INTERFACE I_AlarmControler

PROPERTY Active : REFERENCE TO BOOL
GET
END_GET
END_PROPERTY

PROPERTY ActiveCritical : REFERENCE TO UDINT
GET
END_GET
END_PROPERTY

PROPERTY ActiveError : REFERENCE TO UDINT
GET
END_GET
END_PROPERTY

PROPERTY ActiveInfo : REFERENCE TO UDINT
GET
END_GET
END_PROPERTY

PROPERTY ActiveVerbose : REFERENCE TO UDINT
GET
END_GET
END_PROPERTY

PROPERTY ActiveWarrning : REFERENCE TO UDINT
GET
END_GET
END_PROPERTY

PROPERTY Busy : REFERENCE TO BOOL
GET
END_GET
END_PROPERTY

PROPERTY Error : REFERENCE TO BOOL
GET
END_GET
END_PROPERTY

PROPERTY FileName : STRING
GET
END_GET
SET
END_SET
END_PROPERTY

PROPERTY MaxEvents : UDINT
GET
END_GET
END_PROPERTY

METHOD MR_Abort : BOOL
VAR_INPUT
END_VAR
END_METHOD

METHOD MR_Clear : BOOL
VAR_INPUT
	ipFilter : I_TcEventFilter;
	bResetConfirmation : BOOL;
END_VAR
END_METHOD

METHOD MR_ClearAll : BOOL
VAR_INPUT
	bResetConfirmation : BOOL;
END_VAR
END_METHOD

METHOD MR_Confirm : BOOL
VAR_INPUT
	ipFilter : I_TcEventFilter;
END_VAR
END_METHOD

METHOD MR_ConfirmAll : BOOL
VAR_INPUT
	bResetConfirmation : BOOL;
END_VAR
END_METHOD

METHOD MR_Export : BOOL
VAR_INPUT
END_VAR
END_METHOD

METHOD MR_FirstCycle : BOOL
VAR_INPUT
	sName 		: STRING;
	sFileName 	: STRING;
END_VAR
END_METHOD

METHOD MR_Init : BOOL
VAR_INPUT
END_VAR
END_METHOD

PROPERTY Name : REFERENCE TO STRING
GET
END_GET
END_PROPERTY

PROPERTY State : REFERENCE TO E_AlarmControlerState
GET
END_GET
END_PROPERTY

END_INTERFACE

(* stored: Version 1.1.0.1, ProductVersion 3.1.4024.9
   Itf I_AlarmControler: Id {3984c38c-9915-4540-884b-363753ee2751}
   Property Active: Id {2a8f619a-dd85-4aeb-bd54-75218b29e6bb}
   Get Get: Id {7244eb17-a0e3-4a49-ba5a-69383a84fee4}
   Property ActiveCritical: Id {758ba293-f2f7-4d47-9e34-8110d89d8927}
   Get Get: Id {ae1a4685-6b48-4bfc-82c2-115d2a476243}
   Property ActiveError: Id {48f9ca0b-9866-49b7-accc-404ae7c9e939}
   Get Get: Id {1ba1a4f8-0844-4a46-8a6c-b822060c17f7}
   Property ActiveInfo: Id {2a251e6c-2c4e-482a-b797-0e2508e6bf38}
   Get Get: Id {4218612b-6900-4fa6-afe0-920f58052390}
   Property ActiveVerbose: Id {5b9a0796-635d-416f-ba46-d5c640db2ded}
   Get Get: Id {3f4fe3fe-c087-4d8b-8d77-5f643c999c29}
   Property ActiveWarrning: Id {552e917b-cd99-4c94-a87a-6e8e70ca89ec}
   Get Get: Id {93c7cfff-45a6-4023-a2ac-3d1251be6bbf}
   Property Busy: Id {b836a67d-2552-4e21-997a-9a9a6029707a}
   Get Get: Id {eb22ea72-734c-4002-94b0-ad7d457c7a6b}
   Property Error: Id {e3c05109-7618-42b7-845a-160143d2084c}
   Get Get: Id {fef87d4d-a59e-48de-8beb-4fd0e886ee58}
   Property FileName: Id {abe38245-2d5b-4d79-b04c-c2bd675a9bfe}
   Get Get: Id {29c4f576-e6be-4479-96c8-73e201d0f90e}
   Set Set: Id {1e9518f0-79cd-4c75-96c8-3c5f097bb238}
   Property MaxEvents: Id {1dce21ec-acef-44e1-ba9b-92dc627ccf4a}
   Get Get: Id {89757b0c-eb9e-43b6-8573-57c94d69727a}
   Method MR_Abort: Id {53768c67-5562-4247-933b-2ec4b9184ce8}
   Method MR_Clear: Id {51f02b3f-5314-41b8-a632-d10b698c0672}
   Method MR_ClearAll: Id {ed2ce2c6-09a4-42ab-9464-3b9b5c735f9e}
   Method MR_Confirm: Id {2b6f42c7-602b-443b-ab59-dc82df534d7a}
   Method MR_ConfirmAll: Id {c10c0b48-c0bc-407e-8610-ad5fd9e119ae}
   Method MR_Export: Id {5cb74265-045e-4734-ba05-e937c2a6dab3}
   Method MR_FirstCycle: Id {28463785-51b8-4d36-8e5a-2e273fc8dc05}
   Method MR_Init: Id {bc3cc481-3de9-40b1-9bcc-b187364c9e60}
   Property Name: Id {2099f0ca-50ae-4c8a-8977-c1e3870033b8}
   Get Get: Id {b92729ea-bbee-4cc7-97e9-b3ffbdbbdd81}
   Property State: Id {9eb36b5e-723b-4f4c-b13d-2dda186b7e7e}
   Get Get: Id {cb6a9fe9-39d4-4eda-b999-991d10da0f3a} *)
